// Mitsubishi GX Works2 project: 3sec, Conveyor ON   PLC: FX1N/FX1NC

PROGRAM MAIN
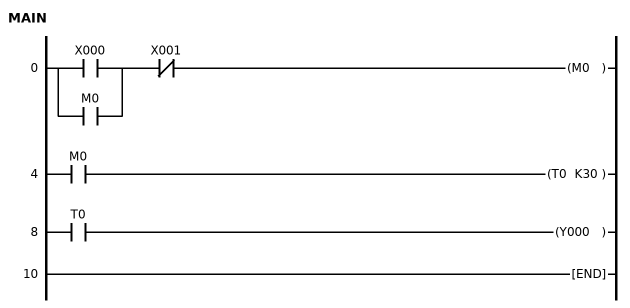
0     LD      X000
      OR      M0
      ANI     X001
      OUT     M0
4     LD      M0
      OUT     T0 K30
8     LD      T0
      OUT     Y000
10    END
END_PROGRAM
